TYPE T_FolderPath : STRING[100];
END_TYPE

(* stored: Version 1.1.0.1
   DUT T_FolderPath: Id {7cbd837c-3240-4cd8-bb89-5cf2d0a63a8e} *)
